(* Logix 5000 project; controller TrayLoader_EnSG vendor 1 type 14 code 156 rev 32.11; software revision 32.02 *)

TASK MainTask (continuous, watchdog 500 ms) : MainProgram

MODULES
   Local : vendor 1 type 14 code 156 (Compact 0, rev 32.11)
      DI2 : 1769-IQ32 (Compact 2, rev 3.1, Input RPI 20 ms)
      DI1 : 1769-IQ32 (Compact 1, rev 3.1, Input RPI 20 ms)
      DI3 : 1769-IQ32 (Compact 3, rev 3.1, Input RPI 20 ms)
      DO2 : vendor 1 type 7 code 73 (Compact 5, rev 3.1, Output RPI 20 ms)
      DO1 : vendor 1 type 7 code 73 (Compact 4, rev 3.1, Output RPI 20 ms)
      PF525_UpLift : PowerFlex 525-EENET (Ethernet 172.20.10.12, rev 5.2, Output RPI 20 ms)
      Feeder : vendor 1 type 37 code 29 (Ethernet 172.20.10.14, rev 2.1, MotionDiagnostics RPI 1 ms, MotionSync RPI 6 ms)
      Tray : 2097-V34PR5-LM (Ethernet 172.20.10.13, rev 2.1, MotionSync RPI 1 ms, MotionDiagnostics RPI 1 ms)
      DemoTray : vendor 1 type 37 code 28 (Ethernet 172.20.10.17, rev 2.1, MotionSync RPI 6 ms, MotionDiagnostics RPI 1 ms)
END_MODULES

VAR_GLOBAL   (* controller tags *)
   Alarm_reedSw : BOOL;
   Auto : BOOL := 1;
   auto_resumeFeeder : BOOL;
   clutch_t : TIMER := (PRE := 500, ACC := 500, EN := 1, DN := 1);
   corr_elapsedTrayPos : DINT := -317;
   ct_lifter_safety : BOOL;
   ct_safety1 : BOOL;   // safety contact
   ct_safety2 : BOOL;
   cycle_t : TIMER := (PRE := 200);
   DecelDelay_t : TIMER := (PRE := 2);
   DecelVal : DINT := 54;
   delta_TrayActualPos : DINT := 121;
   dummy1 : BOOL;
   dummy10 : BOOL;
   dummy11 : BOOL;
   dummy2 : BOOL;
   dummy6 : BOOL;
   dummy7 : BOOL;
   dummy8 : BOOL := 1;
   dummy9 : BOOL;
   elapsedTrayPos : DINT;
   enableCheckingMsg : MESSAGE;
        MessageParameters(ServiceCode := 16#0010, LocalElement := EnableInputChecking, ...)
   enableHwOvertravelMsg : MESSAGE;
        MessageParameters(ServiceCode := 16#0010, LocalElement := EnableInputChecking, ...)
   EnableInputChecking : DINT;
   Fault : BOOL;
   feed_decel_spd : INT := -12;   // mcd speed
   Feed_st : INT;
   FeedConvSMC_PC : BOOL;
   feedDela_t : TIMER := (PRE := 100);
   feedDelay : BOOL;
   FeederConvAxis : AXIS_CIP_DRIVE;
   FeedLine : BOOL := 1;
   FeedLine_ons : BOOL;
   feedReload : BOOL;
   feedReload_t : TIMER := (PRE := 50, ACC := 18, EN := 1, TT := 1);
   FeedSpeed : DINT := 30;
   feedWD_t : TIMER := (PRE := 4000);   // Watch Dog Timer on Feeder
   FinishPush : BOOL;
   finishPush_t : TIMER := (PRE := 5);
   finishPush_t0 : TIMER := (PRE := 30);
   firstLine : BOOL;
   firstLine_stat : BOOL;
   FlipInCanReturn : BOOL := 1;
   gotoFirstLine : BOOL;
   hmi_Reset : BOOL;
   hmi_resetTrayCtr : BOOL;
   hmi_setSpeedRef : DINT := 50;
   hmi_setSpeedRef100 : INT := 5000;
   Idle_Delay : TIMER := (PRE := 100);
   JogPulse_m : BOOL := 1;
   JogTime : TIMER := (PRE := 100);
   lastActualPosUnit : DINT := -259472;
   lineCtr : INT := 18;
   man_disableUplift : BOOL;
   man_engageClutch : BOOL;
   man_feederReload : BOOL;
   man_feedplank : BOOL;
   man_FeedRailEnd : BOOL;
   man_JogLineDown : BOOL;
   man_JogLineUp : BOOL;
   man_ledRun : BOOL;
   man_ledStart : BOOL;
   man_ledWarning : BOOL;
   man_mot_conv_in0 : BOOL;
   man_mot_conv_in1 : BOOL;
   man_mot_conv_in2 : BOOL;
   man_mot_conv_in3 : BOOL;
   man_mot_conv_in4 : BOOL;
   man_mot_upLiftBrake : BOOL;
   man_nc_ps_exit : BOOL;
   man_ps_vert_upLifter : BOOL := 1;
   man_rs_sv_exit_bot : BOOL := 1;
   man_rs_sv_exit_top : BOOL;
   man_rs_sv_flipperIn_bot : BOOL;
   man_rs_sv_flipperIn_top : BOOL;
   man_serp_top : BOOL;
   man_sol_engageClutch : BOOL;
   man_SrvTrayJogMotorFwd : BOOL;
   man_srvTrayStop : BOOL;
   man_stop_conveyor : BOOL;
   man_sv_exit : BOOL;
   man_sv_flipperIn : BOOL := 1;
   man_sv_flipperOut : BOOL;
   man_sv_flipperOut_bot : BOOL;
   man_sv_flipperOut_top : BOOL;
   man_sv_gripper : BOOL;
   man_sv_gripperArm : BOOL;
   man_sv_tray_in : BOOL;
   man_sv_tray_out : BOOL;
   man_UpLift_forward : BOOL := 1;
   man_UpLift_start : BOOL;
   mot_upLiftBrake : BOOL;
   MotFault : BOOL;
   nc_ls_UpLift_bot : BOOL;
   nc_ls_UpLift_top : BOOL;
   nc_ps_exit : BOOL;   // indicate Full exit qeue
   nc_ps_tray_in_ons : BOOL;
   nc_ps_tray_out : BOOL;   // nc tray load bottom
   nc_ps_trayFeed_top : BOOL := 1;
   nc_ps_trayFeed_top_ons : BOOL := 1;
   nc_px_tray_in : BOOL;   // Servo bucket detected
   nc_px_trayFeed_bot : BOOL;   // ps tray before feeder
   nc_px_trayFeed_bot_ons : BOOL;
   nc_px_UpLift_bot : BOOL;
   nc_px_UpLift_top : BOOL;
   negStepPulse : DINT := -120;
   no_ps_FeedPlankHome : BOOL := 1;
   no_ps_FeedPlankHome_inv_ons : BOOL;
   no_ps_FeedPlankHome_ons : BOOL;
   no_ps_FeedRailDecel : BOOL;
   no_ps_FeedRailEndEven : BOOL;   // ps on end of FeederRail
   no_ps_FeedRailEndOdd : BOOL;
   no_ps_flipperIn : BOOL;
   no_ps_posTransfer : BOOL;
   no_ps_Serp_bot : BOOL := 1;   // ps Serpentine Bottom
   no_ps_Serp_top : BOOL;   // ps serpentine top
   no_ps_tray_in_top : BOOL := 1;
   no_ps_vert_upLifter : BOOL := 1;
   no_sw_pressure : BOOL;
   ons2 : DINT;
   ons3 : DINT;
   ons4 : INT := 32;
   ons6 : DINT := 579;
   ons7 : DINT;
   pauseFeeder : BOOL;
   pb_Emergency : BOOL;
   pb_safetyReset : BOOL;
   pb_Start : BOOL;
   pb_Stop : BOOL;
   probe0 : BOOL;
   ps_flipperIn_t : TIMER := (PRE := 2000);
   ps_flipperIn_tof : TIMER := (PRE := 2000, ACC := 2000, EN := 1, DN := 1);
   ps_serp_top_t : TIMER := (PRE := 1000);
   ps_serp_top_tof : TIMER := (PRE := 1000);
   RailDecel : BOOL;
   ReadyArmToPush : BOOL;
   Recover_UpLift : BOOL;
   ref_elpasedTrayPos : DINT := 1680;
   Reset : BOOL;
   resumeFeeder : BOOL;
   rs_sv_exit_bot : BOOL := 1;
   rs_sv_exit_top : BOOL;
   rs_sv_flipperIn_bot : BOOL;
   rs_sv_flipperIn_top : BOOL := 1;
   rs_sv_flipperOut_bot : BOOL := 1;
   rs_sv_flipperOut_top : BOOL;
   rs_sv_gripArm_bot : BOOL := 1;   // rs pneu gripper arm bottom
   rs_sv_gripArm_top : BOOL;   // rs pneu gripper arm top
   rs_sv_gripper_grip : BOOL;
   rs_sv_gripper_release : BOOL := 1;
   rs_sv_tray_in_bot : BOOL := 1;
   rs_sv_tray_in_bot_ons : BOOL;
   rs_sv_tray_in_top : BOOL;
   rs_sv_tray_in_top_ons : BOOL;
   rs_sv_tray_out_bot : BOOL := 1;
   rs_sv_tray_out_bot_ons : BOOL;
   rs_sv_tray_out_top : BOOL;
   Run : BOOL;
   RunOff_t : TIMER := (PRE := 500, EN := 1, TT := 1);
   RunOn_t : TIMER := (PRE := 500);
   Safety : BOOL;
   safety_sys_ok : BOOL;
   serp_top_t_pre : DINT := 1000;
   serp_top_tof_pre : DINT := 1000;
   servo_on_t : TIMER := (PRE := 1000, ACC := 1000, EN := 1, DN := 1);
   ServoEndRun : BOOL;
   ServoEndRun_ons : BOOL;
   ServoEndRunPulse : BOOL;
   ServoGroup : MOTION_GROUP;
   sol_engage_t : TIMER := (PRE := 800);
   sol_engageClutch : BOOL;
   SrvTrayJogMot : BOOL;
   SrvTrayStep : BOOL;   // Servo Tray Step down
   SrvTrayStep_t : TIMER := (PRE := 100, ACC := 101, EN := 1, DN := 1);
   SrvTrayStop : BOOL;
   StartSpeed : DINT := 30;
   stepback_t : TIMER := (PRE := 2000);
   stepPulse : DINT := 120;
   stepPulseAct : DINT := 120;
   sv_exit : BOOL;
   sv_flipperIn : BOOL;
   sv_flipperOut : BOOL;
   sv_flipperOut_bot : BOOL;
   sv_flipperOut_top : BOOL;
   sv_gripper : BOOL;
   sv_gripper_bot : BOOL;   // pneu gripper
   sv_gripper_top : BOOL;
   sv_gripperArm : BOOL;
   sv_tray_in : BOOL;
   sv_tray_out : BOOL;
   sw_doorFront : BOOL;
   sw_doorSideA : BOOL;
   sw_doorSideB : BOOL;
   sw_doorTop : BOOL;
   sysStop : BOOL;
   Tmr1 : TIMER := (PRE := 3000);
   tmr_feedinterval : TIMER := (PRE := 300);
   TmrUpLift_top : TIMER := (PRE := 1000);
   torque_limit : BOOL;
   total_tray : DINT := 2;
   Transfer_Pos : BOOL;
   TrayAxis : AXIS_CIP_DRIVE;
   TrayClear : BOOL;
   trayOnFlipperIn : BOOL;
   TraySrvBreakU : BOOL;
   TrayWComp_m : BOOL;   // Compensator mode
   UpLift_2base : BOOL;
   Uplift_idle : BOOL;
   UpLift_stepBack : BOOL;
   UpLift_Up : BOOL := 1;
   Warning : BOOL;
END_VAR

PROGRAM MainProgram   (* main routine MainRoutine *)
VAR
   blink1s : BOOL;
   Bottom_Wait_Pos : BOOL;
   Emergency : BOOL;
   Empty_Wait_Pos : BOOL;
   feeder_finish : BOOL;
   Feeder_st : INT := 2;
   feederReload : BOOL;   // trayLoad step down enabled
   FeedMotionCtrl : MOTION_INSTRUCTION := (FLAGS := 570425344, DN := 1, STATUS := 2, STATE := 1);
   modRes : INT;
   mot_conv_in : INT;   // Conveyor Motor
   no_ps_conv : INT;   // Conveyor Proxi no
   oddEven : BOOL;
   ons : DINT := -1776287743;
   ons5 : INT;
   Pos_Search : BOOL;
   PushLine : BOOL;
   SrvGoHome : BOOL;
   srvMASRTray : BOOL;
   SrvMoveType : DINT := 1;
   t1s_tof : TIMER := (PRE := 1000);
   t1s_ton : TIMER := (PRE := 1000, ACC := 142, EN := 1, TT := 1);
   tmr_reedSw : TIMER := (PRE := 10000);
   TrayAxis_pos : DINT := 120;   // servo position increment
   TrayMotionCtrl : MOTION_INSTRUCTION := (FLAGS := 704643072, DN := 1, PC := 1);
   UpLift_forward : BOOL;
   UpLift_start : BOOL := 1;
   UpLift_stop : BOOL := 1;
END_VAR

ROUTINE _00_Diagnostics   (* ladder *)
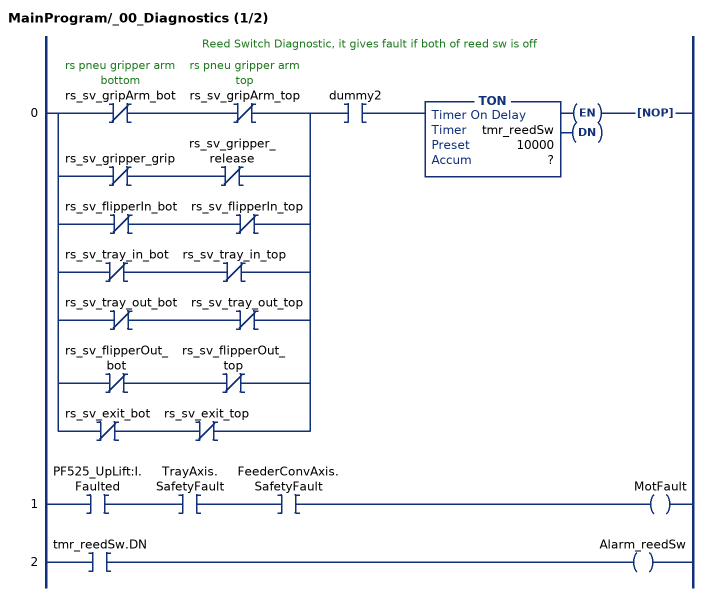
   // Reed Switch Diagnostic, it gives fault if both of reed sw is off
   0: [XIO(rs_sv_gripArm_bot) XIO(rs_sv_gripArm_top) ,XIO(rs_sv_gripper_grip) XIO(rs_sv_gripper_release) ,XIO(rs_sv_flipperIn_bot) XIO(rs_sv_flipperIn_top) ,XIO(rs_sv_tray_in_bot) XIO(rs_sv_tray_in_top) ,XIO(rs_sv_tray_out_bot) XIO(rs_sv_tray_out_top) ,XIO(rs_sv_flipperOut_bot) XIO(rs_sv_flipperOut_top) ,XIO(rs_sv_exit_bot) XIO(rs_sv_exit_top) ]XIC(dummy2)TON(tmr_reedSw,?,?)NOP();
   1: XIC(PF525_UpLift:I.Faulted)XIC(TrayAxis.SafetyFault)XIC(FeederConvAxis.SafetyFault)OTE(MotFault);
   2: XIC(tmr_reedSw.DN)OTE(Alarm_reedSw);
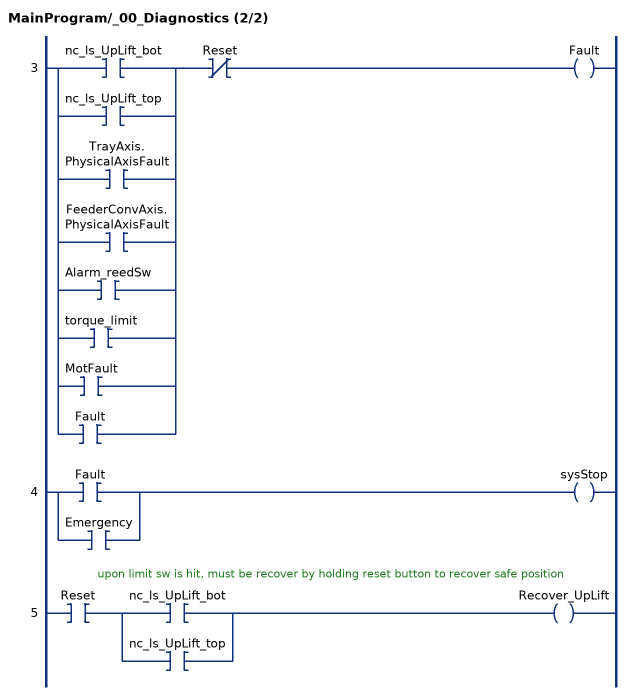
   3: [XIC(nc_ls_UpLift_bot) ,XIC(nc_ls_UpLift_top) ,XIC(TrayAxis.PhysicalAxisFault) ,XIC(FeederConvAxis.PhysicalAxisFault) ,XIC(Alarm_reedSw) ,XIC(torque_limit) ,XIC(MotFault) ,XIC(Fault) ]XIO(Reset)OTE(Fault);
   4: [XIC(Fault) ,XIC(Emergency) ]OTE(sysStop);
   // upon limit sw is hit, must be recover by holding reset button to recover safe position
   5: XIC(Reset)[XIC(nc_ls_UpLift_bot) ,XIC(nc_ls_UpLift_top) ]OTE(Recover_UpLift);
END_ROUTINE

ROUTINE _01_Start   (* ladder *)
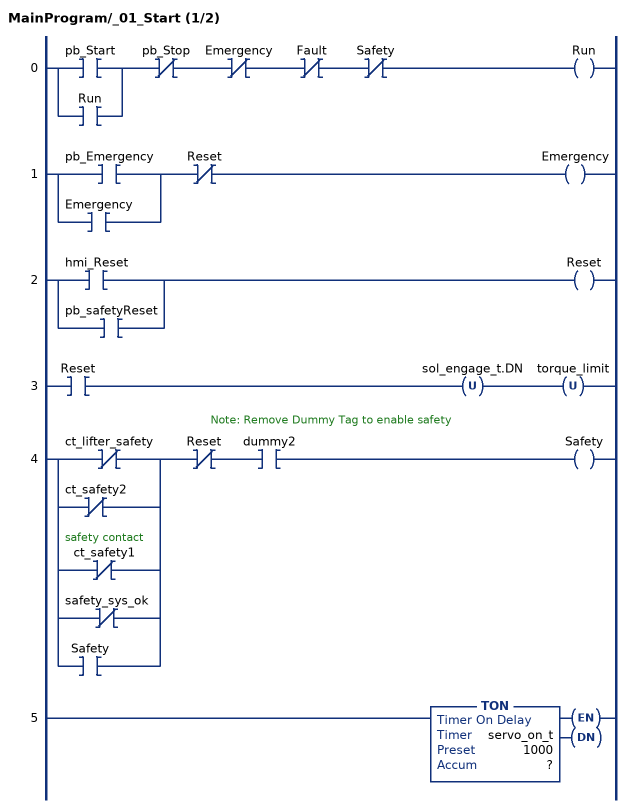
   0: [XIC(pb_Start) ,XIC(Run) ]XIO(pb_Stop)XIO(Emergency)XIO(Fault)XIO(Safety)OTE(Run);
   1: [XIC(pb_Emergency) ,XIC(Emergency) ]XIO(Reset)OTE(Emergency);
   2: [XIC(hmi_Reset) ,XIC(pb_safetyReset) ]OTE(Reset);
   3: XIC(Reset)OTU(sol_engage_t.DN)OTU(torque_limit);
   // Note: Remove Dummy Tag to enable safety
   4: [XIO(ct_lifter_safety) ,XIO(ct_safety2) ,XIO(ct_safety1) ,XIO(safety_sys_ok) ,XIC(Safety) ]XIO(Reset)XIC(dummy2)OTE(Safety);
   5: TON(servo_on_t,?,?);
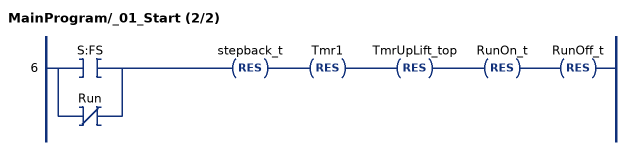
   6: [XIC(S:FS) ,XIO(Run) ]RES(stepback_t)RES(Tmr1)RES(TmrUpLift_top)RES(RunOn_t)RES(RunOff_t);
END_ROUTINE

ROUTINE _02_Inputs   (* ladder *)
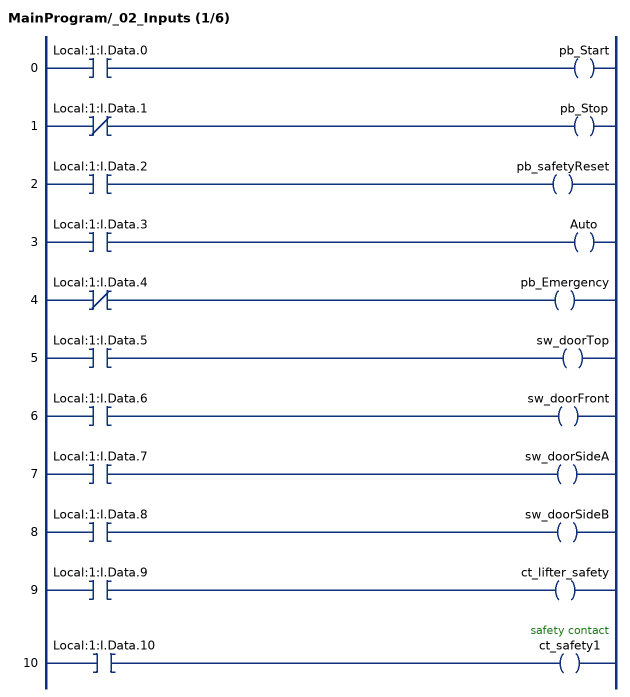
   0: XIC(Local:1:I.Data.0)OTE(pb_Start);
   1: XIO(Local:1:I.Data.1)OTE(pb_Stop);
   2: XIC(Local:1:I.Data.2)OTE(pb_safetyReset);
   3: XIC(Local:1:I.Data.3)OTE(Auto);
   4: XIO(Local:1:I.Data.4)OTE(pb_Emergency);
   5: XIC(Local:1:I.Data.5)OTE(sw_doorTop);
   6: XIC(Local:1:I.Data.6)OTE(sw_doorFront);
   7: XIC(Local:1:I.Data.7)OTE(sw_doorSideA);
   8: XIC(Local:1:I.Data.8)OTE(sw_doorSideB);
   9: XIC(Local:1:I.Data.9)OTE(ct_lifter_safety);
   10: XIC(Local:1:I.Data.10)OTE(ct_safety1);
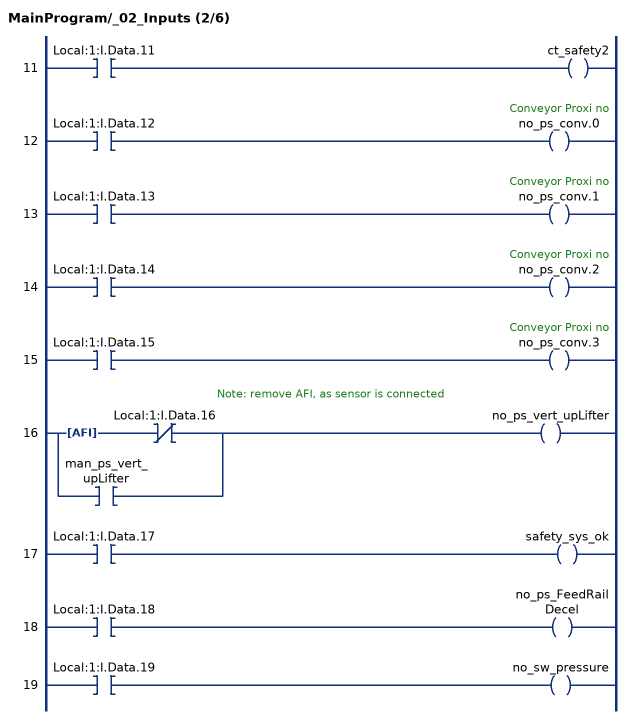
   11: XIC(Local:1:I.Data.11)OTE(ct_safety2);
   12: XIC(Local:1:I.Data.12)OTE(no_ps_conv.0);
   13: XIC(Local:1:I.Data.13)OTE(no_ps_conv.1);
   14: XIC(Local:1:I.Data.14)OTE(no_ps_conv.2);
   15: XIC(Local:1:I.Data.15)OTE(no_ps_conv.3);
   // Note: remove AFI, as sensor is connected
   16: [AFI() XIO(Local:1:I.Data.16) ,XIC(man_ps_vert_upLifter) ]OTE(no_ps_vert_upLifter);
   17: XIC(Local:1:I.Data.17)OTE(safety_sys_ok);
   18: XIC(Local:1:I.Data.18)OTE(no_ps_FeedRailDecel);
   19: XIC(Local:1:I.Data.19)OTE(no_sw_pressure);
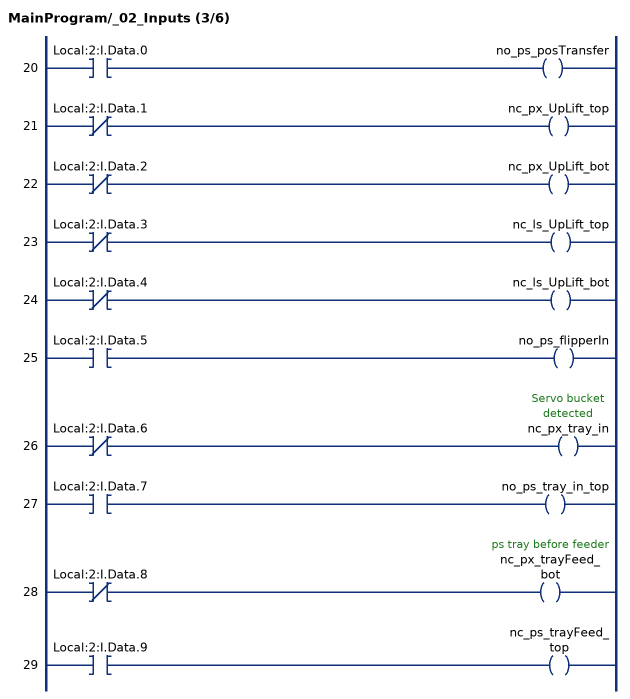
   20: XIC(Local:2:I.Data.0)OTE(no_ps_posTransfer);
   21: XIO(Local:2:I.Data.1)OTE(nc_px_UpLift_top);
   22: XIO(Local:2:I.Data.2)OTE(nc_px_UpLift_bot);
   23: XIO(Local:2:I.Data.3)OTE(nc_ls_UpLift_top);
   24: XIO(Local:2:I.Data.4)OTE(nc_ls_UpLift_bot);
   25: XIC(Local:2:I.Data.5)OTE(no_ps_flipperIn);
   26: XIO(Local:2:I.Data.6)OTE(nc_px_tray_in);
   27: XIC(Local:2:I.Data.7)OTE(no_ps_tray_in_top);
   28: XIO(Local:2:I.Data.8)OTE(nc_px_trayFeed_bot);
   29: XIC(Local:2:I.Data.9)OTE(nc_ps_trayFeed_top);
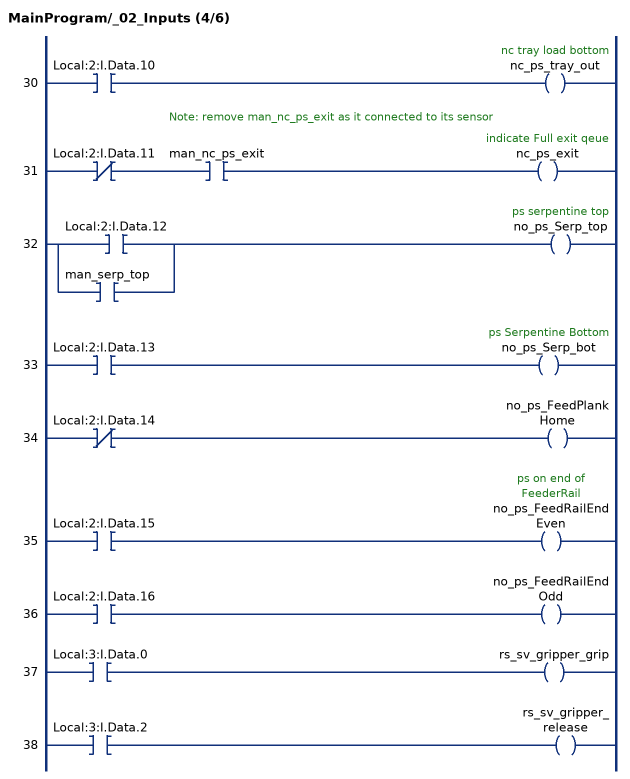
   30: XIC(Local:2:I.Data.10)OTE(nc_ps_tray_out);
   // Note: remove man_nc_ps_exit as it connected to its sensor
   31: XIO(Local:2:I.Data.11)XIC(man_nc_ps_exit)OTE(nc_ps_exit);
   32: [XIC(Local:2:I.Data.12) ,XIC(man_serp_top) ]OTE(no_ps_Serp_top);
   33: XIC(Local:2:I.Data.13)OTE(no_ps_Serp_bot);
   34: XIO(Local:2:I.Data.14)OTE(no_ps_FeedPlankHome);
   35: XIC(Local:2:I.Data.15)OTE(no_ps_FeedRailEndEven);
   36: XIC(Local:2:I.Data.16)OTE(no_ps_FeedRailEndOdd);
   37: XIC(Local:3:I.Data.0)OTE(rs_sv_gripper_grip);
   38: XIC(Local:3:I.Data.2)OTE(rs_sv_gripper_release);
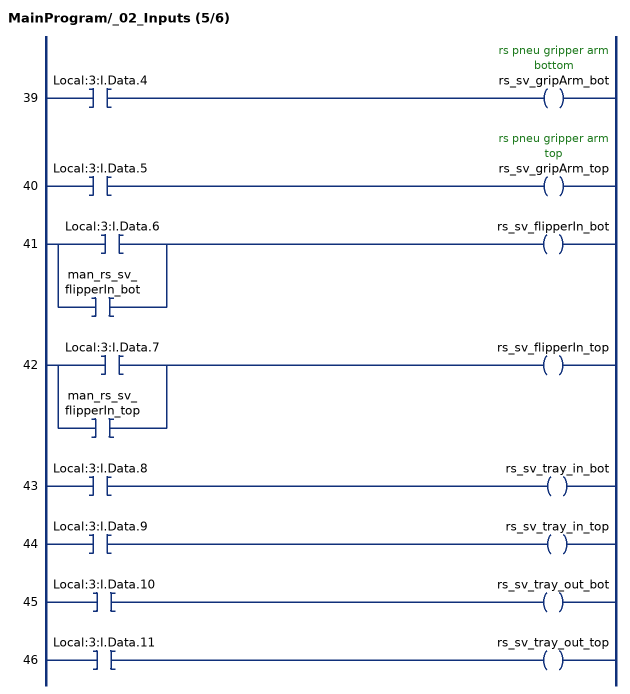
   39: XIC(Local:3:I.Data.4)OTE(rs_sv_gripArm_bot);
   40: XIC(Local:3:I.Data.5)OTE(rs_sv_gripArm_top);
   41: [XIC(Local:3:I.Data.6) ,XIC(man_rs_sv_flipperIn_bot) ]OTE(rs_sv_flipperIn_bot);
   42: [XIC(Local:3:I.Data.7) ,XIC(man_rs_sv_flipperIn_top) ]OTE(rs_sv_flipperIn_top);
   43: XIC(Local:3:I.Data.8)OTE(rs_sv_tray_in_bot);
   44: XIC(Local:3:I.Data.9)OTE(rs_sv_tray_in_top);
   45: XIC(Local:3:I.Data.10)OTE(rs_sv_tray_out_bot);
   46: XIC(Local:3:I.Data.11)OTE(rs_sv_tray_out_top);
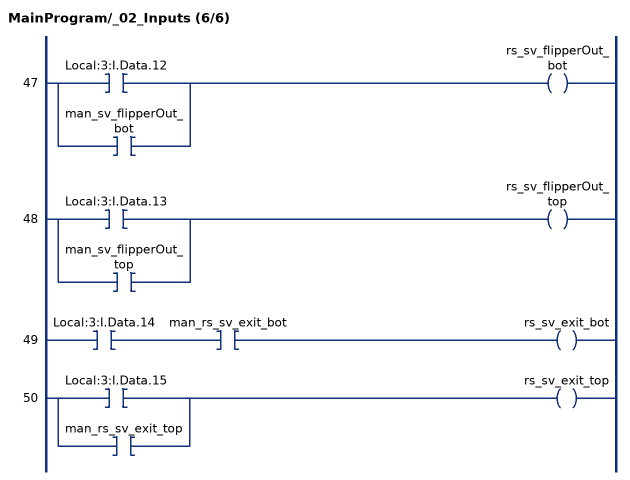
   47: [XIC(Local:3:I.Data.12) ,XIC(man_sv_flipperOut_bot) ]OTE(rs_sv_flipperOut_bot);
   48: [XIC(Local:3:I.Data.13) ,XIC(man_sv_flipperOut_top) ]OTE(rs_sv_flipperOut_top);
   49: XIC(Local:3:I.Data.14)XIC(man_rs_sv_exit_bot)OTE(rs_sv_exit_bot);
   50: [XIC(Local:3:I.Data.15) ,XIC(man_rs_sv_exit_top) ]OTE(rs_sv_exit_top);
END_ROUTINE

ROUTINE _03_Conveyor   (* ladder *)
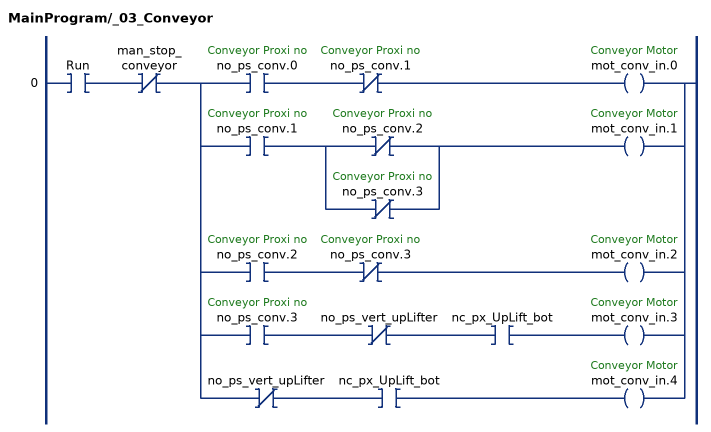
   0: XIC(Run)XIO(man_stop_conveyor)[XIC(no_ps_conv.0) XIO(no_ps_conv.1) OTE(mot_conv_in.0) ,XIC(no_ps_conv.1) [XIO(no_ps_conv.2) ,XIO(no_ps_conv.3) ] OTE(mot_conv_in.1) ,XIC(no_ps_conv.2) XIO(no_ps_conv.3) OTE(mot_conv_in.2) ,XIC(no_ps_conv.3) XIO(no_ps_vert_upLifter) XIC(nc_px_UpLift_bot) OTE(mot_conv_in.3) ,XIO(no_ps_vert_upLifter) XIC(nc_px_UpLift_bot) OTE(mot_conv_in.4) ];
END_ROUTINE

ROUTINE _04_Dispenser   (* ladder *)
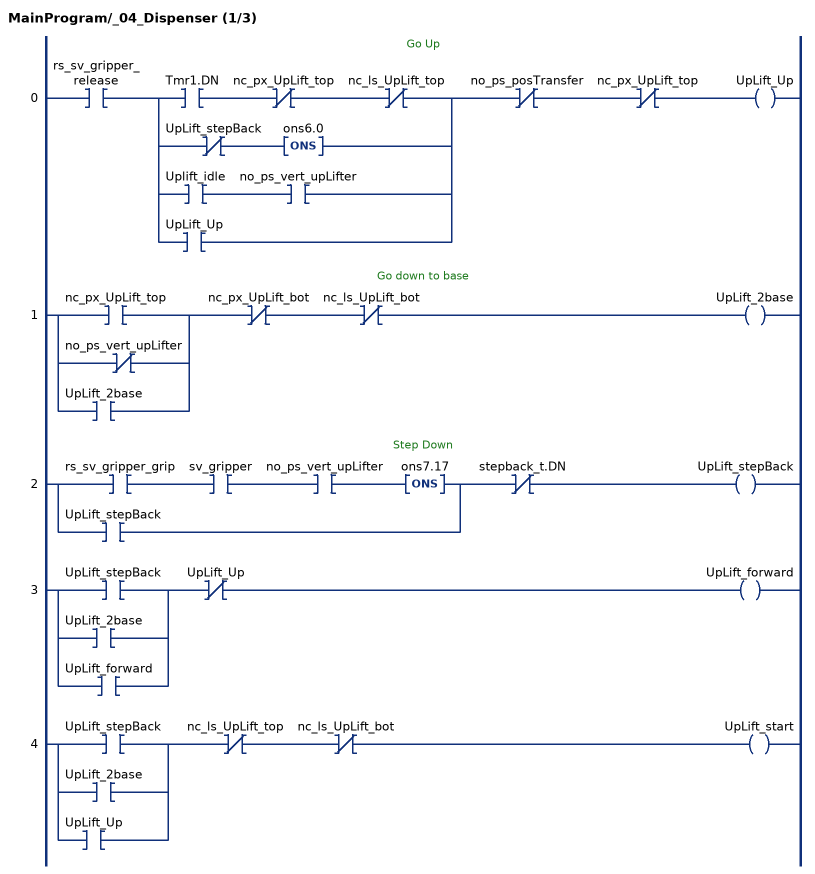
   // Go Up
   0: XIC(rs_sv_gripper_release)[XIC(Tmr1.DN) XIO(nc_px_UpLift_top) XIO(nc_ls_UpLift_top) ,XIO(UpLift_stepBack) ONS(ons6.0) ,XIC(Uplift_idle) XIC(no_ps_vert_upLifter) ,XIC(UpLift_Up) ]XIO(no_ps_posTransfer)XIO(nc_px_UpLift_top)OTE(UpLift_Up);
   // Go down to base
   1: [[XIC(nc_px_UpLift_top) ,XIO(no_ps_vert_upLifter) ] ,XIC(UpLift_2base) ]XIO(nc_px_UpLift_bot)XIO(nc_ls_UpLift_bot)OTE(UpLift_2base);
   // Step Down
   2: [XIC(rs_sv_gripper_grip) XIC(sv_gripper) XIC(no_ps_vert_upLifter) ONS(ons7.17) ,XIC(UpLift_stepBack) ]XIO(stepback_t.DN)OTE(UpLift_stepBack);
   3: [XIC(UpLift_stepBack) ,XIC(UpLift_2base) ,XIC(UpLift_forward) ]XIO(UpLift_Up)OTE(UpLift_forward);
   4: [XIC(UpLift_stepBack) ,XIC(UpLift_2base) ,XIC(UpLift_Up) ]XIO(nc_ls_UpLift_top)XIO(nc_ls_UpLift_bot)OTE(UpLift_start);
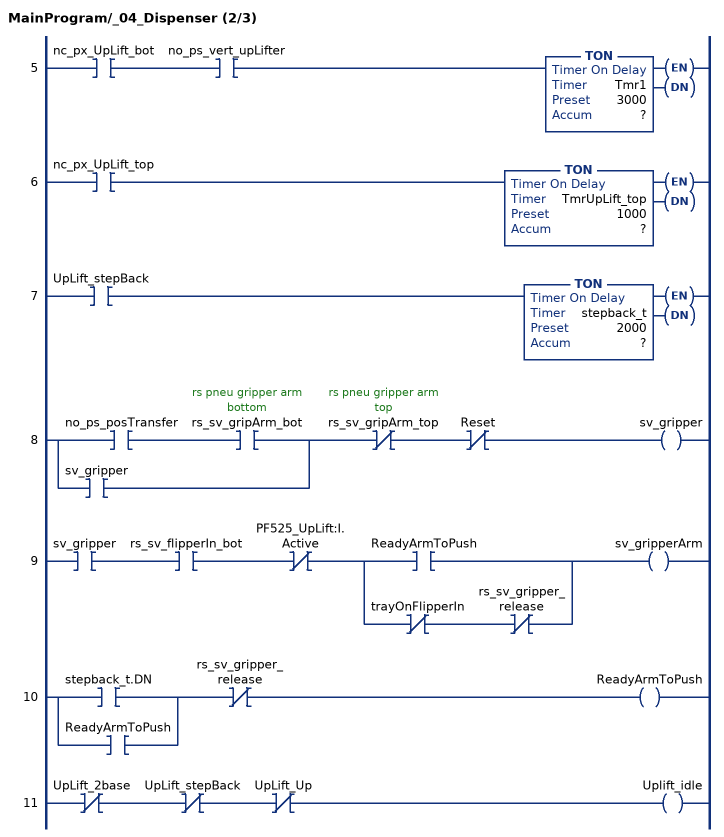
   5: XIC(nc_px_UpLift_bot)XIC(no_ps_vert_upLifter)TON(Tmr1,?,?);
   6: XIC(nc_px_UpLift_top)TON(TmrUpLift_top,?,?);
   7: XIC(UpLift_stepBack)TON(stepback_t,?,?);
   8: [XIC(no_ps_posTransfer) XIC(rs_sv_gripArm_bot) ,XIC(sv_gripper) ]XIO(rs_sv_gripArm_top)XIO(Reset)OTE(sv_gripper);
   9: XIC(sv_gripper)XIC(rs_sv_flipperIn_bot)XIO(PF525_UpLift:I.Active)[XIC(ReadyArmToPush) ,XIO(trayOnFlipperIn) XIO(rs_sv_gripper_release) ]OTE(sv_gripperArm);
   10: [XIC(stepback_t.DN) ,XIC(ReadyArmToPush) ]XIO(rs_sv_gripper_release)OTE(ReadyArmToPush);
   11: XIO(UpLift_2base)XIO(UpLift_stepBack)XIO(UpLift_Up)OTE(Uplift_idle);
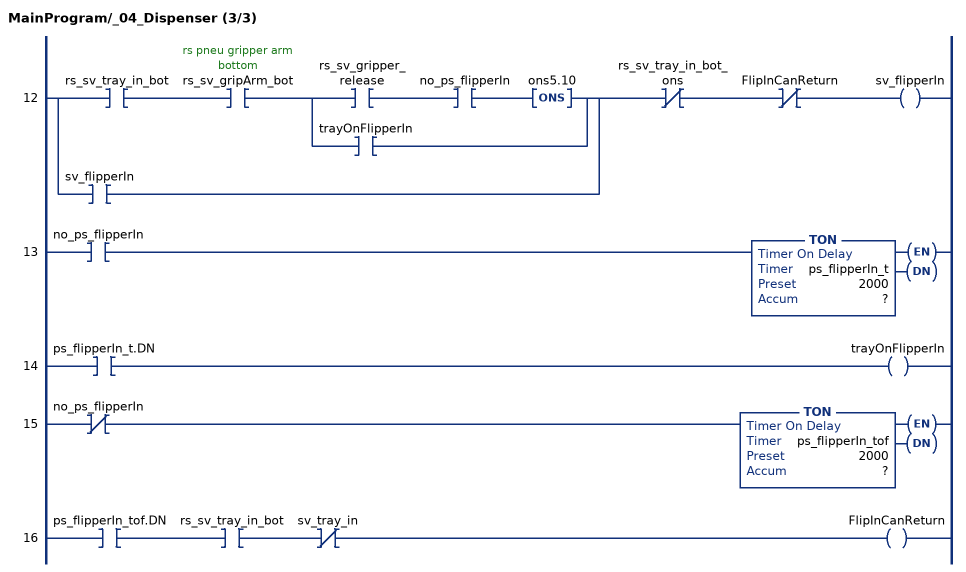
   12: [XIC(rs_sv_tray_in_bot) XIC(rs_sv_gripArm_bot) [XIC(rs_sv_gripper_release) XIC(no_ps_flipperIn) ONS(ons5.10) ,XIC(trayOnFlipperIn) ] ,XIC(sv_flipperIn) ]XIO(rs_sv_tray_in_bot_ons)XIO(FlipInCanReturn)OTE(sv_flipperIn);
   13: XIC(no_ps_flipperIn)TON(ps_flipperIn_t,?,?);
   14: XIC(ps_flipperIn_t.DN)OTE(trayOnFlipperIn);
   15: XIO(no_ps_flipperIn)TON(ps_flipperIn_tof,?,?);
   16: XIC(ps_flipperIn_tof.DN)XIC(rs_sv_tray_in_bot)XIO(sv_tray_in)OTE(FlipInCanReturn);
END_ROUTINE

ROUTINE _04_Run   (* ladder *)
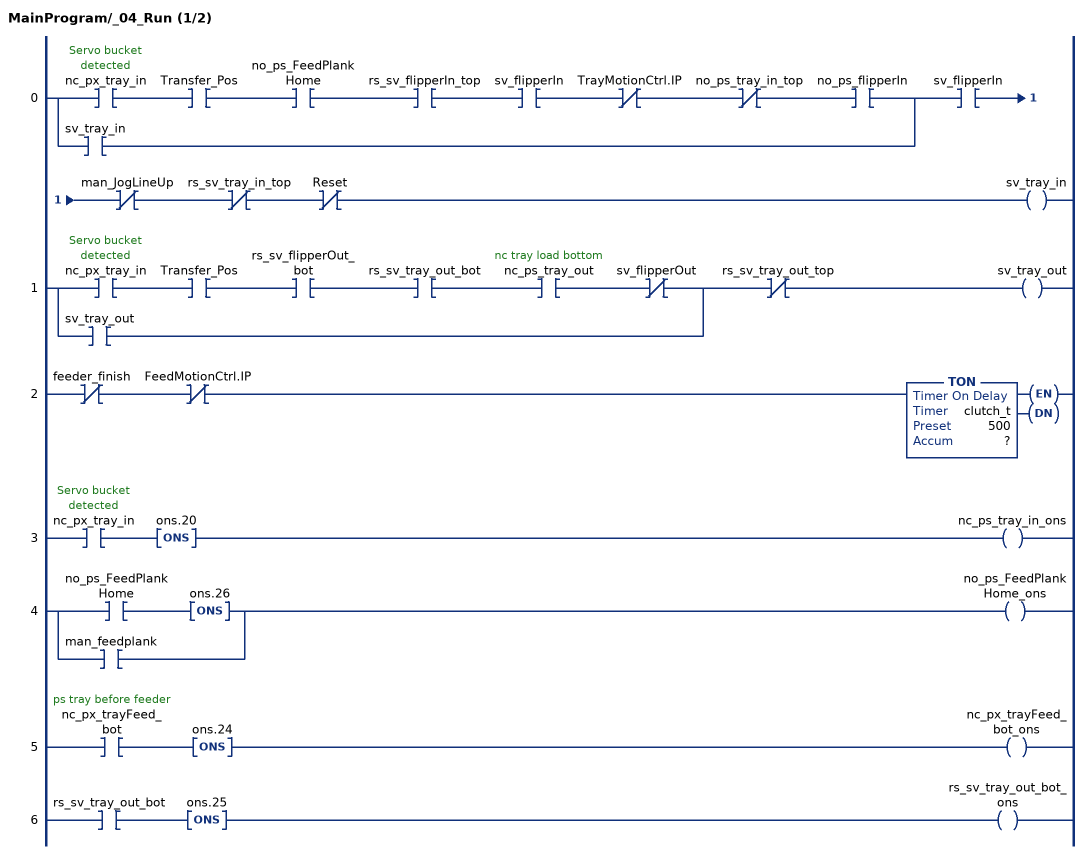
   0: [XIC(nc_px_tray_in) XIC(Transfer_Pos) XIC(no_ps_FeedPlankHome) XIC(rs_sv_flipperIn_top) XIC(sv_flipperIn) XIO(TrayMotionCtrl.IP) XIO(no_ps_tray_in_top) XIC(no_ps_flipperIn) ,XIC(sv_tray_in) ]XIC(sv_flipperIn)XIO(man_JogLineUp)XIO(rs_sv_tray_in_top)XIO(Reset)OTE(sv_tray_in);
   1: [XIC(nc_px_tray_in) XIC(Transfer_Pos) XIC(rs_sv_flipperOut_bot) XIC(rs_sv_tray_out_bot) XIC(nc_ps_tray_out) XIO(sv_flipperOut) ,XIC(sv_tray_out) ]XIO(rs_sv_tray_out_top)OTE(sv_tray_out);
   2: XIO(feeder_finish)XIO(FeedMotionCtrl.IP)TON(clutch_t,?,?);
   3: XIC(nc_px_tray_in)ONS(ons.20)OTE(nc_ps_tray_in_ons);
   4: [XIC(no_ps_FeedPlankHome) ONS(ons.26) ,XIC(man_feedplank) ]OTE(no_ps_FeedPlankHome_ons);
   5: XIC(nc_px_trayFeed_bot)ONS(ons.24)OTE(nc_px_trayFeed_bot_ons);
   6: XIC(rs_sv_tray_out_bot)ONS(ons.25)OTE(rs_sv_tray_out_bot_ons);
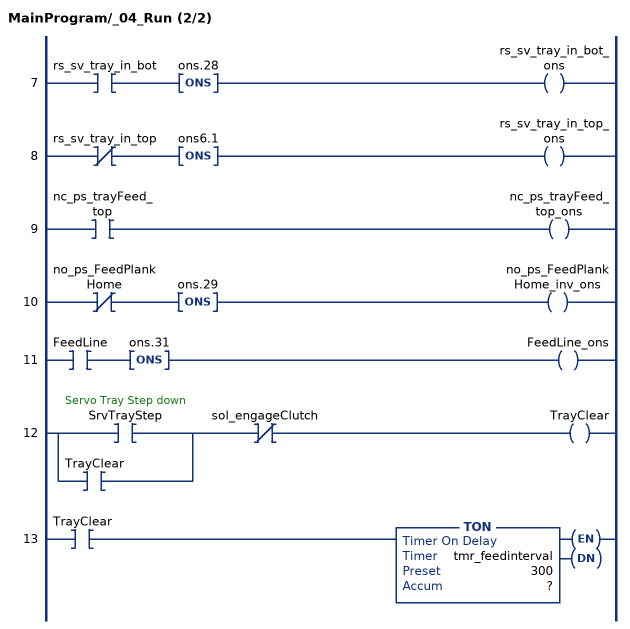
   7: XIC(rs_sv_tray_in_bot)ONS(ons.28)OTE(rs_sv_tray_in_bot_ons);
   8: XIO(rs_sv_tray_in_top)ONS(ons6.1)OTE(rs_sv_tray_in_top_ons);
   9: XIC(nc_ps_trayFeed_top)OTE(nc_ps_trayFeed_top_ons);
   10: XIO(no_ps_FeedPlankHome)ONS(ons.29)OTE(no_ps_FeedPlankHome_inv_ons);
   11: XIC(FeedLine)ONS(ons.31)OTE(FeedLine_ons);
   12: [XIC(SrvTrayStep) ,XIC(TrayClear) ]XIO(sol_engageClutch)OTE(TrayClear);
   13: XIC(TrayClear)TON(tmr_feedinterval,?,?);
END_ROUTINE

ROUTINE _05_Feeder   (* ladder *)
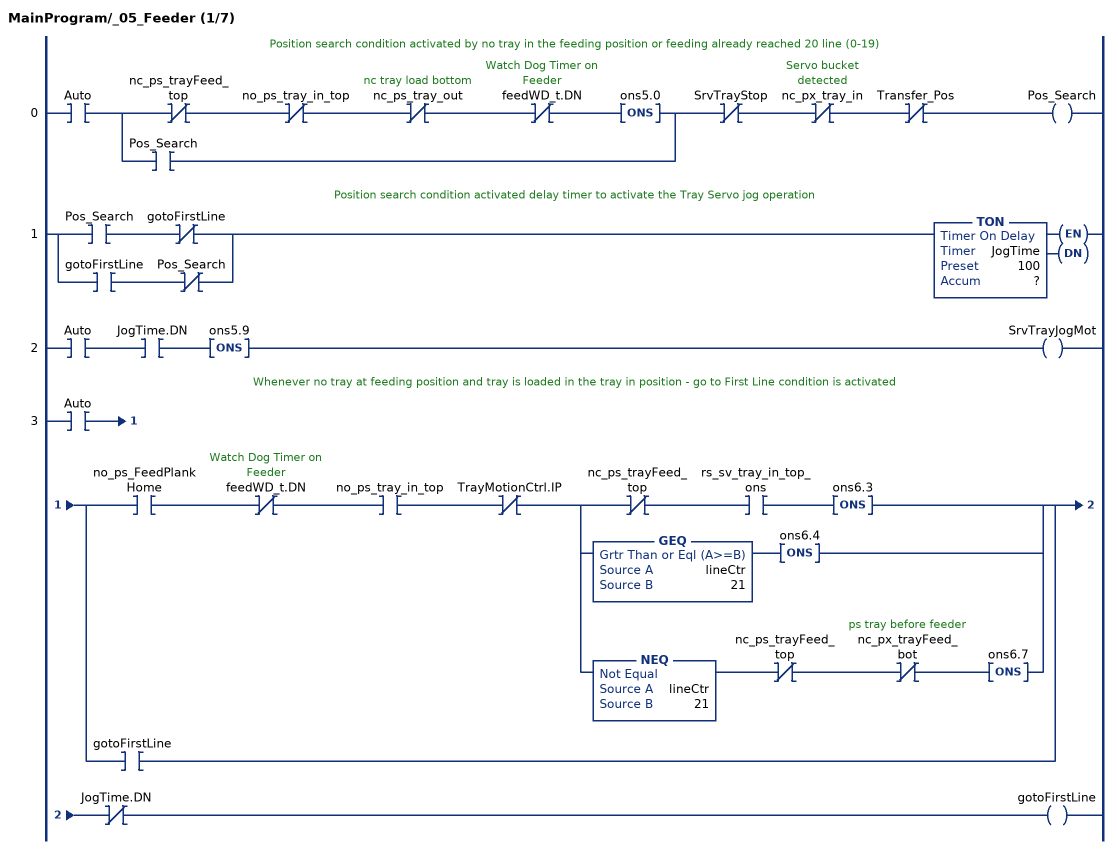
   // Position search condition activated by no tray in the feeding position or feeding already reached 20 line (0-19)
   0: XIC(Auto)[XIO(nc_ps_trayFeed_top) XIO(no_ps_tray_in_top) XIO(nc_ps_tray_out) XIO(feedWD_t.DN) ONS(ons5.0) ,XIC(Pos_Search) ]XIO(SrvTrayStop)XIO(nc_px_tray_in)XIO(Transfer_Pos)OTE(Pos_Search);
   // Position search condition activated delay timer to activate the Tray Servo jog operation
   1: [XIC(Pos_Search) XIO(gotoFirstLine) ,XIC(gotoFirstLine) XIO(Pos_Search) ]TON(JogTime,?,?);
   2: XIC(Auto)XIC(JogTime.DN)ONS(ons5.9)OTE(SrvTrayJogMot);
   // Whenever no tray at feeding position and tray is loaded in the tray in position - go to First Line condition is activated
   3: XIC(Auto)[XIC(no_ps_FeedPlankHome) XIO(feedWD_t.DN) XIC(no_ps_tray_in_top) XIO(TrayMotionCtrl.IP) [XIO(nc_ps_trayFeed_top) XIC(rs_sv_tray_in_top_ons) ONS(ons6.3) ,GEQ(lineCtr,21) ONS(ons6.4) ,NEQ(lineCtr,21) XIO(nc_ps_trayFeed_top) XIO(nc_px_trayFeed_bot) ONS(ons6.7) ] ,XIC(gotoFirstLine) ]XIO(JogTime.DN)OTE(gotoFirstLine);
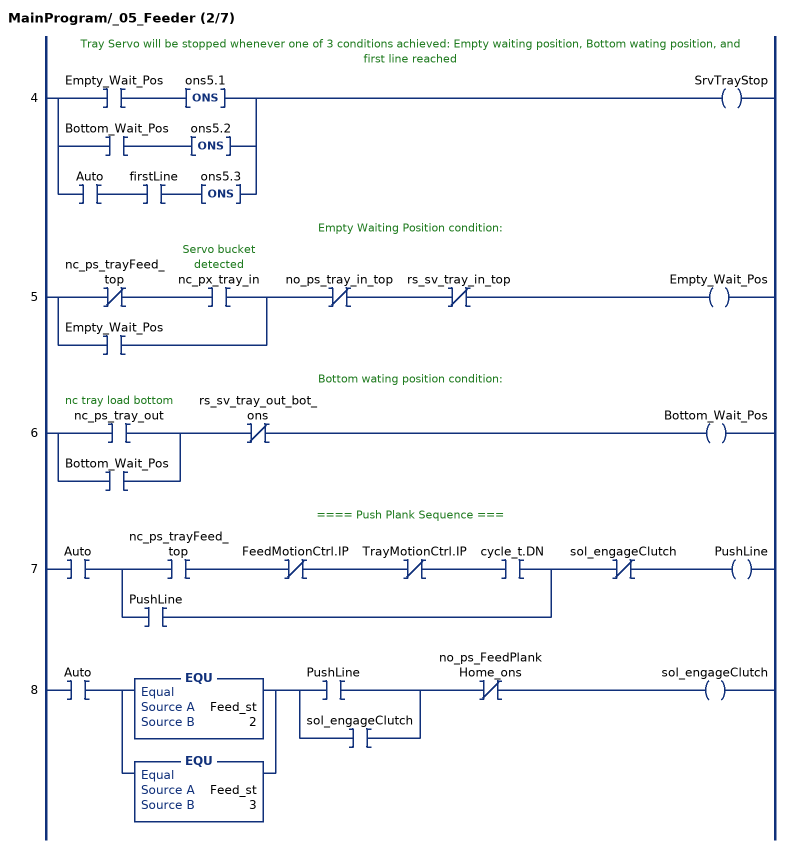
   // Tray Servo will be stopped whenever one of 3 conditions achieved: Empty waiting position, Bottom wating position, and first line reached
   4: [XIC(Empty_Wait_Pos) ONS(ons5.1) ,XIC(Bottom_Wait_Pos) ONS(ons5.2) ,XIC(Auto) XIC(firstLine) ONS(ons5.3) ]OTE(SrvTrayStop);
   // Empty Waiting Position condition:
   5: [XIO(nc_ps_trayFeed_top) XIC(nc_px_tray_in) ,XIC(Empty_Wait_Pos) ]XIO(no_ps_tray_in_top)XIO(rs_sv_tray_in_top)OTE(Empty_Wait_Pos);
   // Bottom wating position condition:
   6: [XIC(nc_ps_tray_out) ,XIC(Bottom_Wait_Pos) ]XIO(rs_sv_tray_out_bot_ons)OTE(Bottom_Wait_Pos);
   // ==== Push Plank Sequence ===
   7: XIC(Auto)[XIC(nc_ps_trayFeed_top) XIO(FeedMotionCtrl.IP) XIO(TrayMotionCtrl.IP) XIC(cycle_t.DN) ,XIC(PushLine) ]XIO(sol_engageClutch)OTE(PushLine);
   8: XIC(Auto)[EQU(Feed_st,2) ,EQU(Feed_st,3) ][XIC(PushLine) ,XIC(sol_engageClutch) ]XIO(no_ps_FeedPlankHome_ons)OTE(sol_engageClutch);
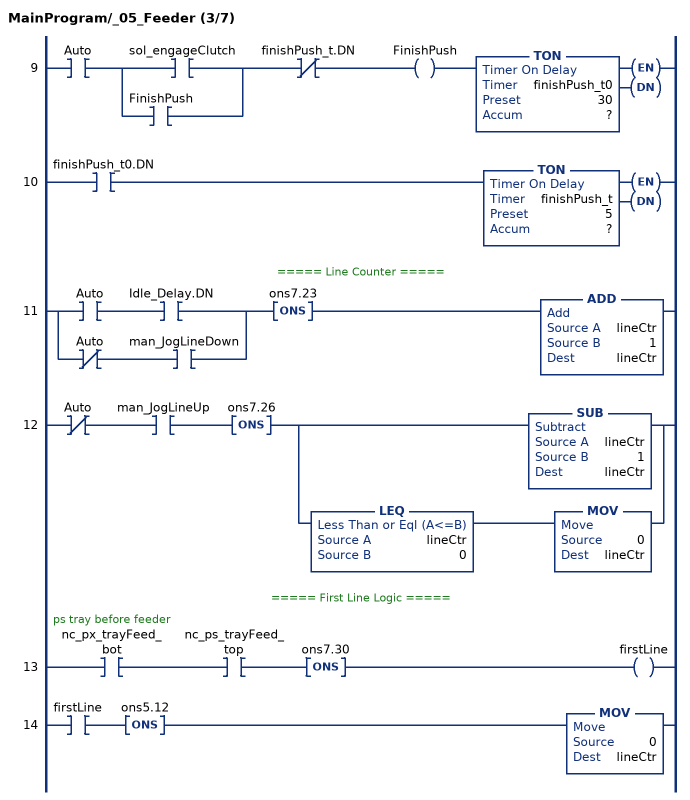
   9: XIC(Auto)[XIC(sol_engageClutch) ,XIC(FinishPush) ]XIO(finishPush_t.DN)OTE(FinishPush)TON(finishPush_t0,?,?);
   10: XIC(finishPush_t0.DN)TON(finishPush_t,?,?);
   // ===== Line Counter =====
   11: [XIC(Auto) XIC(Idle_Delay.DN) ,XIO(Auto) XIC(man_JogLineDown) ]ONS(ons7.23)ADD(lineCtr,1,lineCtr);
   12: XIO(Auto)XIC(man_JogLineUp)ONS(ons7.26)[SUB(lineCtr,1,lineCtr) ,LEQ(lineCtr,0) MOV(0,lineCtr) ];
   // ===== First Line Logic =====
   13: XIC(nc_px_trayFeed_bot)XIC(nc_ps_trayFeed_top)ONS(ons7.30)OTE(firstLine);
   14: XIC(firstLine)ONS(ons5.12)MOV(0,lineCtr);
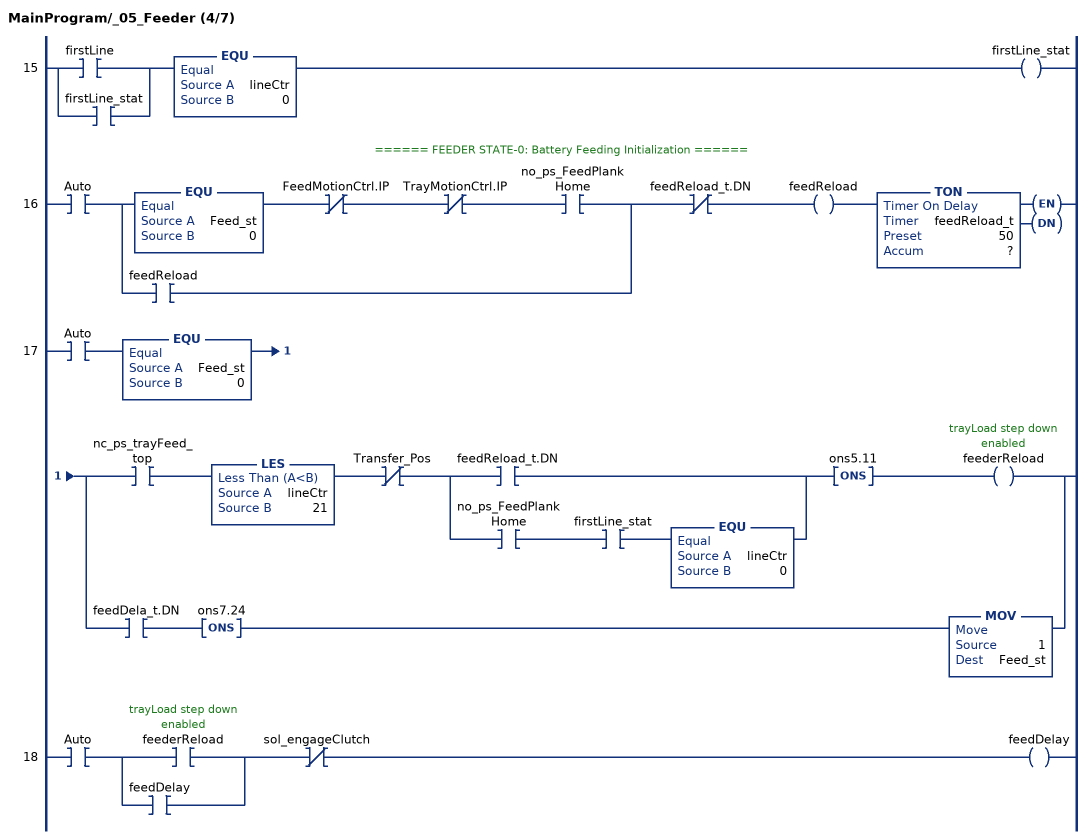
   15: [XIC(firstLine) ,XIC(firstLine_stat) ]EQU(lineCtr,0)OTE(firstLine_stat);
   // ====== FEEDER STATE-0: Battery Feeding Initialization ======
   16: XIC(Auto)[EQU(Feed_st,0) XIO(FeedMotionCtrl.IP) XIO(TrayMotionCtrl.IP) XIC(no_ps_FeedPlankHome) ,XIC(feedReload) ]XIO(feedReload_t.DN)OTE(feedReload)TON(feedReload_t,?,?);
   17: XIC(Auto)EQU(Feed_st,0)[XIC(nc_ps_trayFeed_top) LES(lineCtr,21) XIO(Transfer_Pos) [XIC(feedReload_t.DN) ,XIC(no_ps_FeedPlankHome) XIC(firstLine_stat) EQU(lineCtr,0) ] ONS(ons5.11) OTE(feederReload) ,XIC(feedDela_t.DN) ONS(ons7.24) MOV(1,Feed_st) ];
   18: XIC(Auto)[XIC(feederReload) ,XIC(feedDelay) ]XIO(sol_engageClutch)OTE(feedDelay);
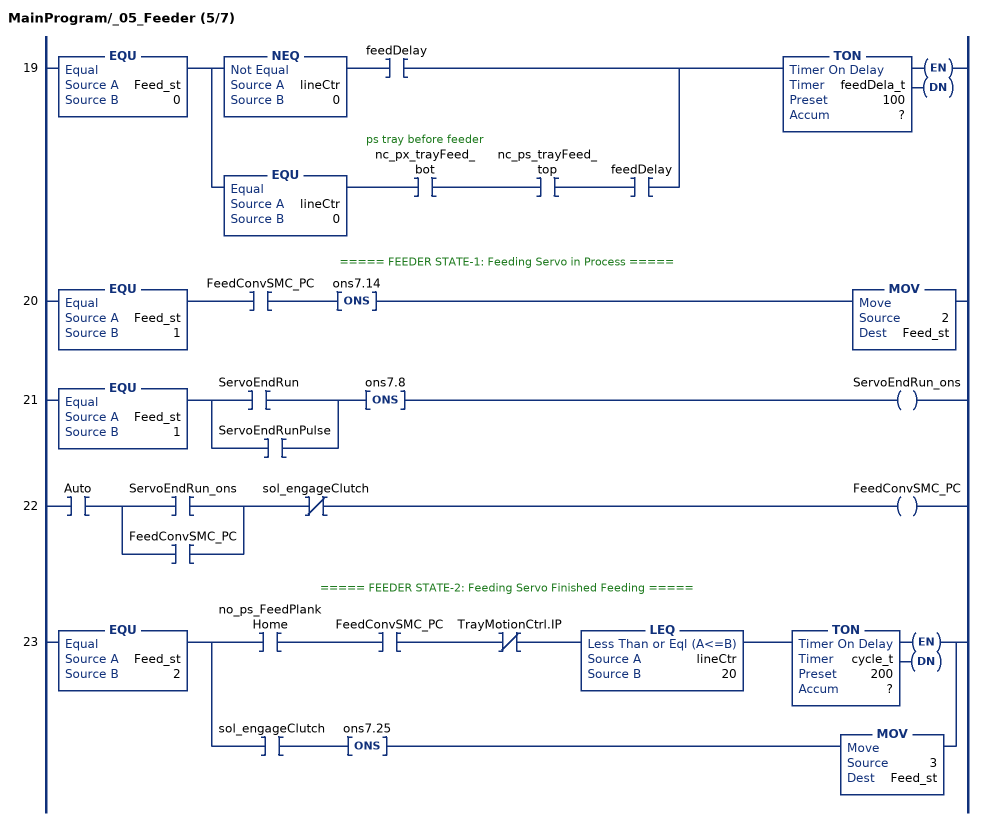
   19: EQU(Feed_st,0)[NEQ(lineCtr,0) XIC(feedDelay) ,EQU(lineCtr,0) XIC(nc_px_trayFeed_bot) XIC(nc_ps_trayFeed_top) XIC(feedDelay) ]TON(feedDela_t,?,?);
   // ===== FEEDER STATE-1: Feeding Servo in Process =====
   20: EQU(Feed_st,1)XIC(FeedConvSMC_PC)ONS(ons7.14)MOV(2,Feed_st);
   21: EQU(Feed_st,1)[XIC(ServoEndRun) ,XIC(ServoEndRunPulse) ]ONS(ons7.8)OTE(ServoEndRun_ons);
   22: XIC(Auto)[XIC(ServoEndRun_ons) ,XIC(FeedConvSMC_PC) ]XIO(sol_engageClutch)OTE(FeedConvSMC_PC);
   // ===== FEEDER STATE-2: Feeding Servo Finished Feeding =====
   23: EQU(Feed_st,2)[XIC(no_ps_FeedPlankHome) XIC(FeedConvSMC_PC) XIO(TrayMotionCtrl.IP) LEQ(lineCtr,20) TON(cycle_t,?,?) ,XIC(sol_engageClutch) ONS(ons7.25) MOV(3,Feed_st) ];
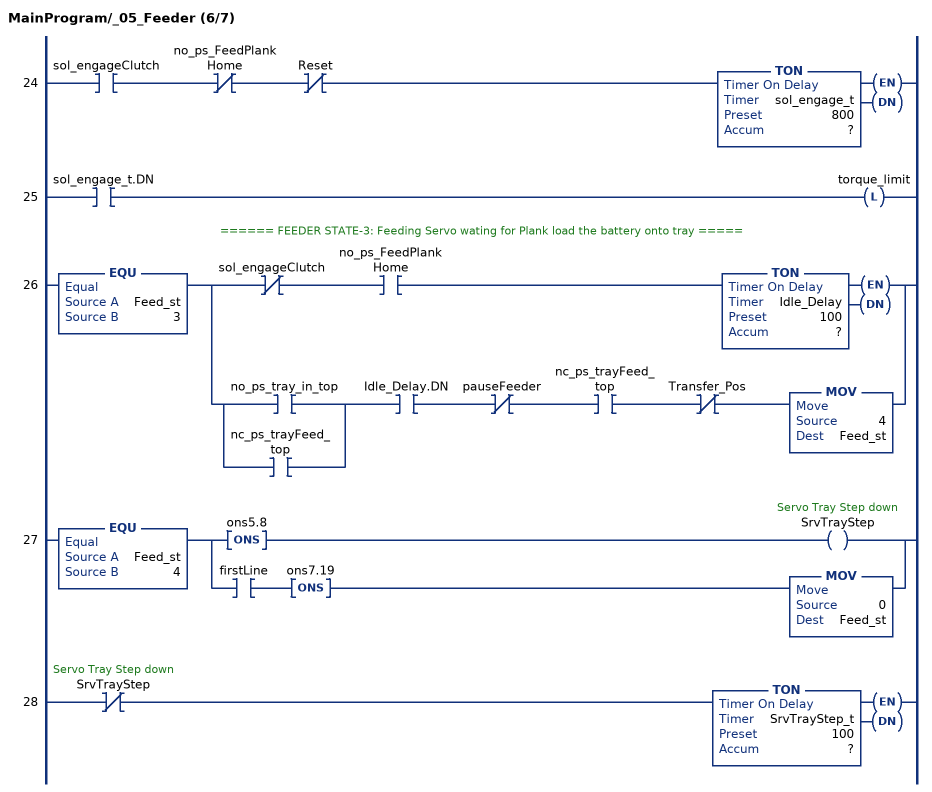
   24: XIC(sol_engageClutch)XIO(no_ps_FeedPlankHome)XIO(Reset)TON(sol_engage_t,?,?);
   25: XIC(sol_engage_t.DN)OTL(torque_limit);
   // ====== FEEDER STATE-3: Feeding Servo wating for Plank load the battery onto tray =====
   26: EQU(Feed_st,3)[XIO(sol_engageClutch) XIC(no_ps_FeedPlankHome) TON(Idle_Delay,?,?) ,[XIC(no_ps_tray_in_top) ,XIC(nc_ps_trayFeed_top) ] XIC(Idle_Delay.DN) XIO(pauseFeeder) XIC(nc_ps_trayFeed_top) XIO(Transfer_Pos) MOV(4,Feed_st) ];
   27: EQU(Feed_st,4)[ONS(ons5.8) OTE(SrvTrayStep) ,XIC(firstLine) ONS(ons7.19) MOV(0,Feed_st) ];
   28: XIO(SrvTrayStep)TON(SrvTrayStep_t,?,?);
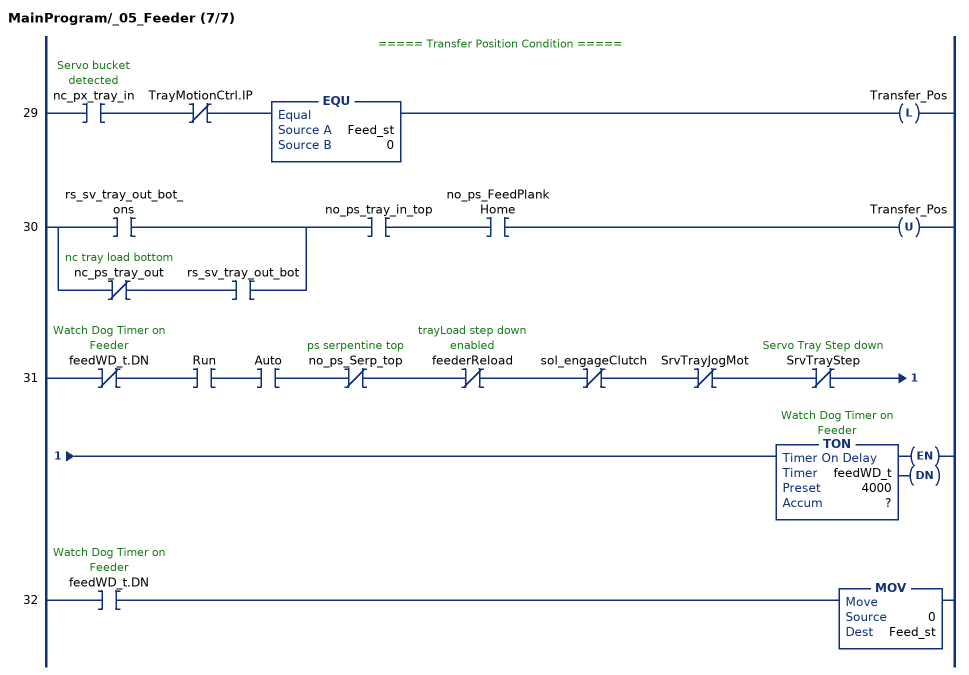
   // ===== Transfer Position Condition =====
   29: XIC(nc_px_tray_in)XIO(TrayMotionCtrl.IP)EQU(Feed_st,0)OTL(Transfer_Pos);
   30: [XIC(rs_sv_tray_out_bot_ons) ,XIO(nc_ps_tray_out) XIC(rs_sv_tray_out_bot) ]XIC(no_ps_tray_in_top)XIC(no_ps_FeedPlankHome)OTU(Transfer_Pos);
   31: XIO(feedWD_t.DN)XIC(Run)XIC(Auto)XIO(no_ps_Serp_top)XIO(feederReload)XIO(sol_engageClutch)XIO(SrvTrayJogMot)XIO(SrvTrayStep)TON(feedWD_t,?,?);
   32: XIC(feedWD_t.DN)MOV(0,Feed_st);
END_ROUTINE
